(* PLC project actuator, TNI-Software ControlBuild 4.00.17 *)
(* stored: creationDateTime 2005-06-20T11:52:37-01:00 *)

FUNCTION_BLOCK cmd_equipment_library.actuator
  VAR_INPUT  (* CB.group=Modes CB.kind=inputVars *)
    autoMode : BOOL := false;  (* CB.mnemonicPatternPropertyName=<SY>_AUTO_<NU> CB.libelle=Automatic mode *)
    manualMode : BOOL := false;  (* CB.mnemonicPatternPropertyName=<SY>_MANU_<NU> CB.libelle=Manual mode *)
  END_VAR
  VAR_INPUT  (* CB.group=Commands CB.kind=inputVars *)
    autoHSCmd : BOOL := false;  (* CB.mnemonicPatternPropertyName=<SY>_CMDGVAUTO_<NU> CB.libelle=Automatic high speed command *)
    autoLSCmd : BOOL := false;  (* CB.mnemonicPatternPropertyName=<SY>_CMDPVAUTO_<NU> CB.libelle=Automatic low speed command *)
  END_VAR
  VAR_INPUT  (* CB.group=PushButtons CB.kind=inputVars *)
    highSpeedPB : BOOL := false;  (* CB.mnemonicPatternPropertyName=<SY>_BPGV_<NU> CB.libelle=High speed pushbutton *)
    lowSpeedPB : BOOL := false;  (* CB.mnemonicPatternPropertyName=<SY>_BPPV_<NU> CB.libelle=Low speed pushbutton *)
    stopPB : BOOL := false;  (* CB.mnemonicPatternPropertyName=<SY>_BPARRET_<NU> CB.libelle=Stop pushbutton *)
  END_VAR
  VAR_INPUT  (* CB.kind=inputVars *)
    generalFault : BOOL := false;  (* CB.mnemonicPatternPropertyName=grlFlt<SY><NU> CB.libelle=General fault of the engine *)
  END_VAR
  VAR_OUTPUT  (* CB.group=Orders CB.kind=outputVars *)
    highSpeedCmd : BOOL := false;  (* CB.mnemonicPatternPropertyName=hSCmd<SY><NU> CB.libelle=High speed command *)
    lowSpeedCmd : BOOL := false;  (* CB.mnemonicPatternPropertyName=lSCmd<SY><NU> CB.libelle=Low speed command *)
  END_VAR

(* LD diagram, written out as Structured Text *)
1:
highSpeedCmd := (autoMode AND autoHSCmd OR manualMode AND (highSpeedPB OR highSpeedCmd) AND NOT lowSpeedPB AND NOT stopPB) AND NOT generalFault;
2:
lowSpeedCmd := (autoMode AND autoLSCmd OR manualMode AND (lowSpeedPB OR lowSpeedCmd) AND NOT highSpeedPB AND NOT stopPB) AND NOT generalFault;
END_FUNCTION_BLOCK
